FUNCTION_BLOCK FB_IODEV_CH_DIGITAL EXTENDS FB_IODEV_CHANNEL
VAR_INPUT
END_VAR
VAR_OUTPUT
END_VAR
VAR
	// Configuration parameters
	// Configured for R/W OPC UA Data Access !!!
	{attribute 'OPC.UA.DA' := '1'}
	{attribute 'OPC.UA.DA.Access' := '3'}
	sLabel_0:	STRING(16)	:= '0';
	{attribute 'OPC.UA.DA' := '1'}
	{attribute 'OPC.UA.DA.Access' := '3'}
	sLabel_1:	STRING(16)	:= '1';
END_VAR

END_FUNCTION_BLOCK

(* stored: Version 1.1.0.1, ProductVersion 3.1.4022.9
   POU FB_IODEV_CH_DIGITAL: Id {608d734d-b375-4889-bba1-588cb9a9f25e}, SpecialFunc None *)
